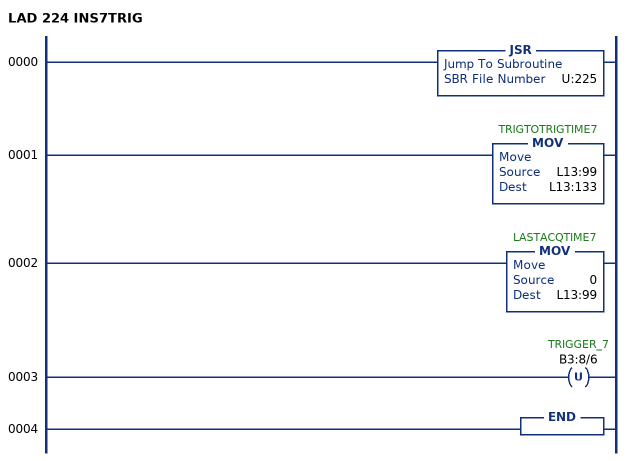
% Rung: 0 %
SOR JSR U:225 EOR
% Rung: 1 %
SOR MOV L13:99 L13:133 EOR
%   L13:99  LASTACQTIME7 %
%   L13:133  TRIGTOTRIGTIME7 %
% Rung: 2 %
SOR MOV 0 L13:99 EOR
%   L13:99  LASTACQTIME7 %
% Rung: 3 %
SOR OTU B3:8/6 EOR
%   B3:8/6  TRIGGER_7 %
% Rung: 4 %
SOR END EOR

LADDER 225 "FIFO7SET"
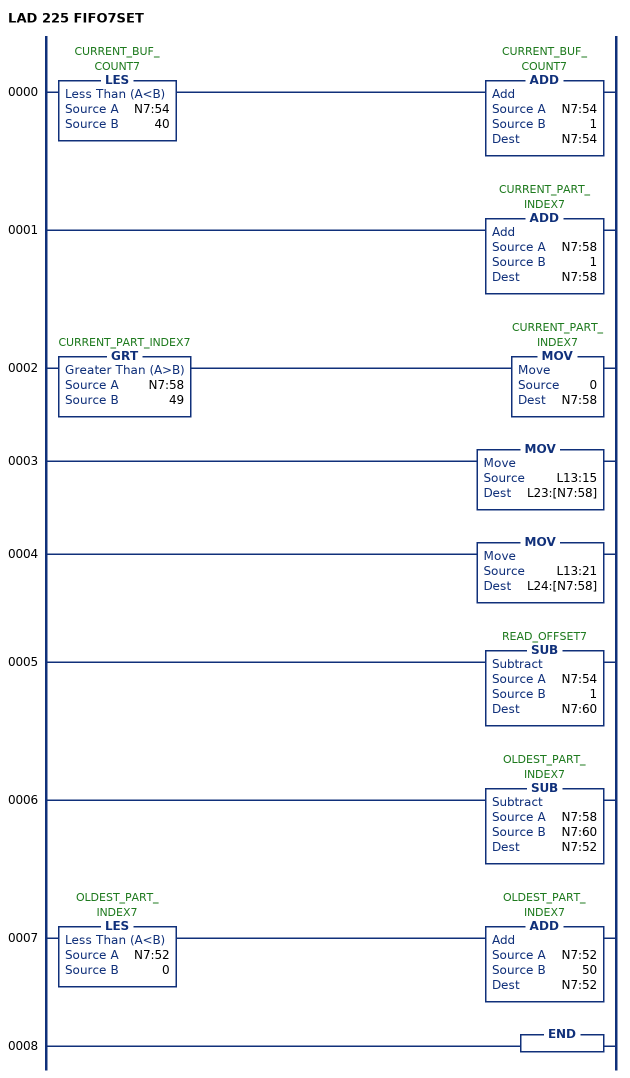
% Rung: 0 %
SOR LES N7:54 40 ADD N7:54 1 N7:54 EOR
%   N7:54  CURRENT_BUF_COUNT7 %
% Rung: 1 %
SOR ADD N7:58 1 N7:58 EOR
%   N7:58  CURRENT_PART_INDEX7 %
% Rung: 2 %
SOR GRT N7:58 49 MOV 0 N7:58 EOR
%   N7:58  CURRENT_PART_INDEX7 %
% Rung: 3 %
SOR MOV L13:15 L23:[N7:58] EOR
%   L13:15  TOP_TIME %
%   N7:58  CURRENT_PART_INDEX7 %
% Rung: 4 %
SOR MOV L13:21 L24:[N7:58] EOR
%   L13:21  TOP_POSITION %
%   N7:58  CURRENT_PART_INDEX7 %
% Rung: 5 %
SOR SUB N7:54 1 N7:60 EOR
%   N7:54  CURRENT_BUF_COUNT7 %
%   N7:60  READ_OFFSET7 %
% Rung: 6 %
SOR SUB N7:58 N7:60 N7:52 EOR
%   N7:58  CURRENT_PART_INDEX7 %
%   N7:60  READ_OFFSET7 %
%   N7:52  OLDEST_PART_INDEX7 %
% Rung: 7 %
SOR LES N7:52 0 ADD N7:52 50 N7:52 EOR
%   N7:52  OLDEST_PART_INDEX7 %
% Rung: 8 %
SOR END EOR

LADDER 226 "FIFO7GET"
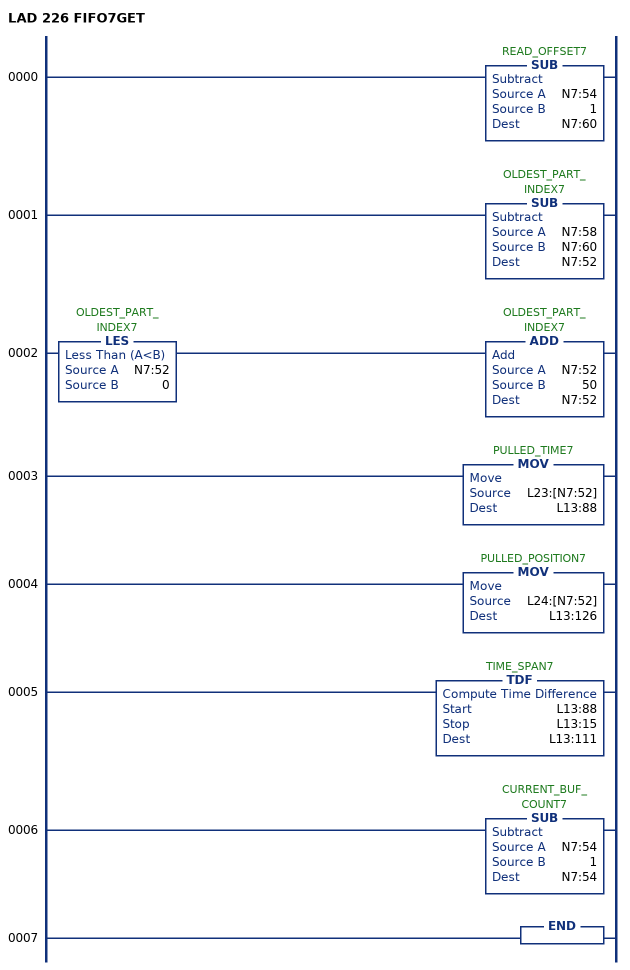
% Rung: 0 %
SOR SUB N7:54 1 N7:60 EOR
%   N7:54  CURRENT_BUF_COUNT7 %
%   N7:60  READ_OFFSET7 %
% Rung: 1 %
SOR SUB N7:58 N7:60 N7:52 EOR
%   N7:58  CURRENT_PART_INDEX7 %
%   N7:60  READ_OFFSET7 %
%   N7:52  OLDEST_PART_INDEX7 %
% Rung: 2 %
SOR LES N7:52 0 ADD N7:52 50 N7:52 EOR
%   N7:52  OLDEST_PART_INDEX7 %
% Rung: 3 %
SOR MOV L23:[N7:52] L13:88 EOR
%   N7:52  OLDEST_PART_INDEX7 %
%   L13:88  PULLED_TIME7 %
% Rung: 4 %
SOR MOV L24:[N7:52] L13:126 EOR
%   N7:52  OLDEST_PART_INDEX7 %
%   L13:126  PULLED_POSITION7 %
% Rung: 5 %
SOR TDF L13:88 L13:15 L13:111 EOR
%   L13:88  PULLED_TIME7 %
%   L13:15  TOP_TIME %
%   L13:111  TIME_SPAN7 %
% Rung: 6 %
SOR SUB N7:54 1 N7:54 EOR
%   N7:54  CURRENT_BUF_COUNT7 %
% Rung: 7 %
SOR END EOR

LADDER 227 "INSDATA7"
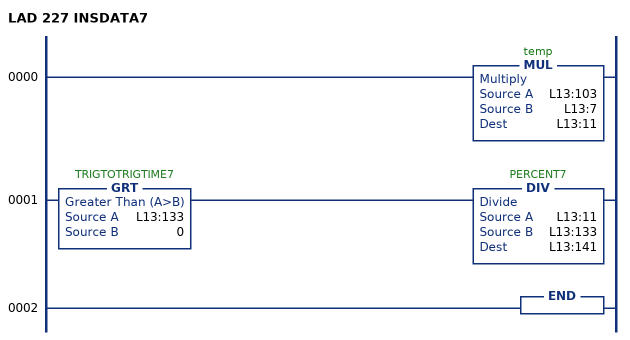
% Rung: 0 %
SOR MUL L13:103 L13:7 L13:11 EOR
%   L13:103  PROCESSTIME7 %
%   L13:7  PERCENT_MULTIPLYER %
%   L13:11  "temp" %
% Rung: 1 %
SOR GRT L13:133 0 DIV L13:11 L13:133 L13:141 EOR
%   L13:133  TRIGTOTRIGTIME7 %
%   L13:11  "temp" %
%   L13:141  PERCENT7 %
% Rung: 2 %
SOR END EOR

LADDER 228 "TESTFAULT7"
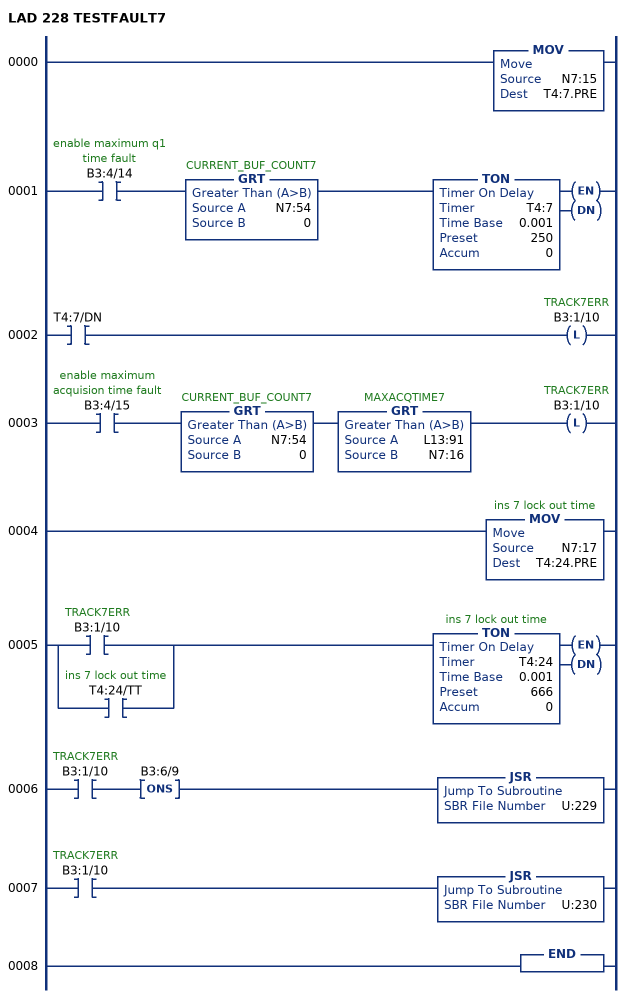
% Rung: 0 %
SOR MOV N7:15 T4:7.PRE EOR
%   N7:15  "max allowed ms time for q to be above 1 if safe fault is used" %
% Rung: 1 %
SOR XIC B3:4/14 GRT N7:54 0 TON T4:7 0.001 250 0 EOR
%   B3:4/14  "enable maximum q1 time fault" %
%   N7:54  CURRENT_BUF_COUNT7 %
% Rung: 2 %
SOR XIC T4:7/DN OTL B3:1/10 EOR
%   B3:1/10  TRACK7ERR %
% Rung: 3 %
SOR XIC B3:4/15 GRT N7:54 0 GRT L13:91 N7:16 OTL B3:1/10 EOR
%   B3:4/15  "enable maximum acquision time fault" %
%   N7:54  CURRENT_BUF_COUNT7 %
%   L13:91  MAXACQTIME7 %
%   N7:16  ACQUIRE_TIME_LIMIT  "maximum of the longest acquire time allowed if maximum acquire time fault is enabled" %
%   B3:1/10  TRACK7ERR %
% Rung: 4 %
SOR MOV N7:17 T4:24.PRE EOR
%   N7:17  "ms time setting to lock out inspection to give all pending images a chance to clear" %
%   T4:24  "ins 7 lock out time" %
% Rung: 5 %
SOR BST XIC B3:1/10 NXB XIC T4:24/TT BND TON T4:24 0.001 666 0 EOR
%   B3:1/10  TRACK7ERR %
%   T4:24  "ins 7 lock out time" %
% Rung: 6 %
SOR XIC B3:1/10 ONS B3:6/9 JSR U:229 EOR
%   B3:1/10  TRACK7ERR %
% Rung: 7 %
SOR XIC B3:1/10 JSR U:230 EOR
%   B3:1/10  TRACK7ERR %
% Rung: 8 %
SOR END EOR

LADDER 229 "INS7FIX1"
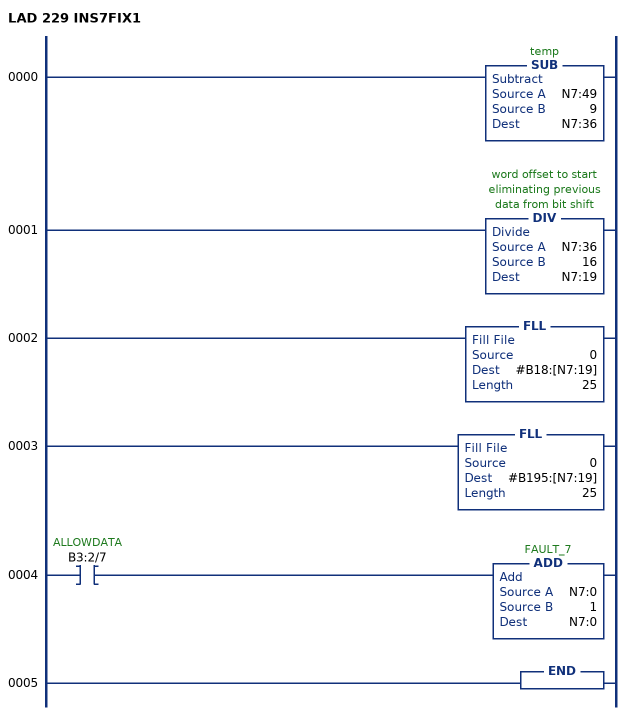
% Rung: 0 %
SOR SUB N7:49 9 N7:36 EOR
%   N7:49  INS_7_TRIG_LOC %
%   N7:36  "temp" %
% Rung: 1 %
SOR DIV N7:36 16 N7:19 EOR
%   N7:36  "temp" %
%   N7:19  "word offset to start eliminating previous data from bit shift" %
% Rung: 2 %
SOR FLL 0 #B18:[N7:19] 25 EOR
%   N7:19  "word offset to start eliminating previous data from bit shift" %
% Rung: 3 %
SOR FLL 0 #B195:[N7:19] 25 EOR
%   N7:19  "word offset to start eliminating previous data from bit shift" %
% Rung: 4 %
SOR XIC B3:2/7 ADD N7:0 1 N7:0 EOR
%   B3:2/7  ALLOWDATA %
%   N7:0  FAULT_7 %
% Rung: 5 %
SOR END EOR

LADDER 230 "INS7FIX2"
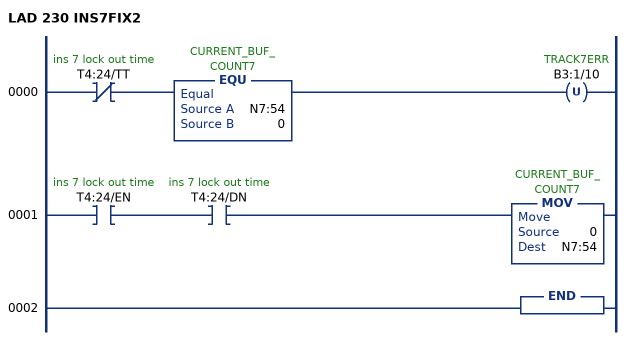
% Rung: 0 %
SOR XIO T4:24/TT EQU N7:54 0 OTU B3:1/10 EOR
%   T4:24  "ins 7 lock out time" %
%   N7:54  CURRENT_BUF_COUNT7 %
%   B3:1/10  TRACK7ERR %
% Rung: 1 %
SOR XIC T4:24/EN XIC T4:24/DN MOV 0 N7:54 EOR
%   T4:24  "ins 7 lock out time" %
%   N7:54  CURRENT_BUF_COUNT7 %
% Rung: 2 %
SOR END EOR

LADDER 232 "INS8"
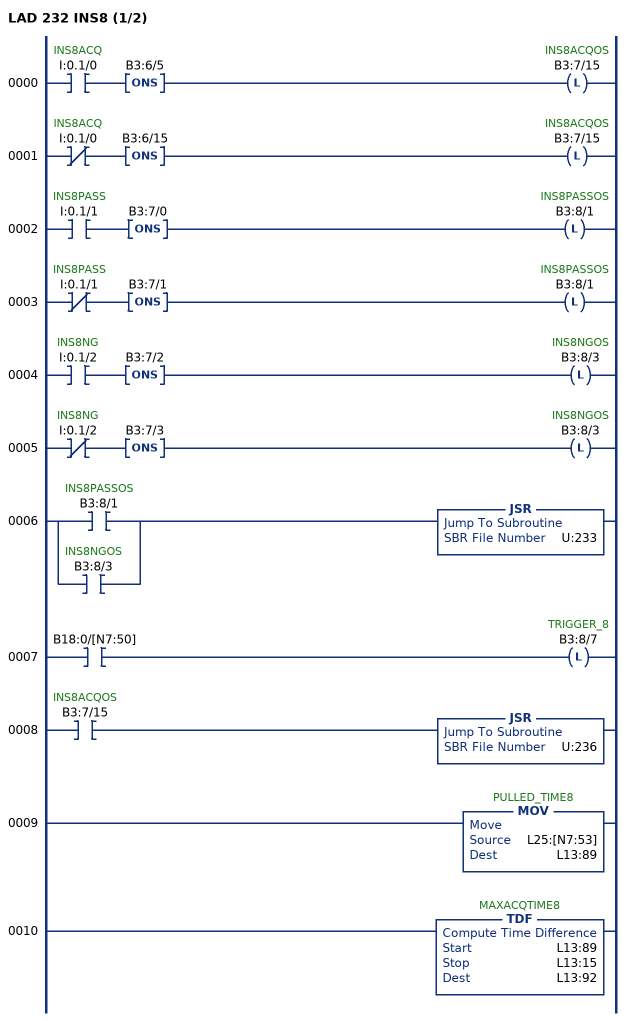
% Rung: 0 %
SOR XIC I:0.1/0 ONS B3:6/5 OTL B3:7/15 EOR
%   I:0.1/0  INS8ACQ %
%   B3:7/15  INS8ACQOS %
% Rung: 1 %
SOR XIO I:0.1/0 ONS B3:6/15 OTL B3:7/15 EOR
%   I:0.1/0  INS8ACQ %
%   B3:7/15  INS8ACQOS %
% Rung: 2 %
SOR XIC I:0.1/1 ONS B3:7/0 OTL B3:8/1 EOR
%   I:0.1/1  INS8PASS %
%   B3:8/1  INS8PASSOS %
% Rung: 3 %
SOR XIO I:0.1/1 ONS B3:7/1 OTL B3:8/1 EOR
%   I:0.1/1  INS8PASS %
%   B3:8/1  INS8PASSOS %
% Rung: 4 %
SOR XIC I:0.1/2 ONS B3:7/2 OTL B3:8/3 EOR
%   I:0.1/2  INS8NG %
%   B3:8/3  INS8NGOS %
% Rung: 5 %
SOR XIO I:0.1/2 ONS B3:7/3 OTL B3:8/3 EOR
%   I:0.1/2  INS8NG %
%   B3:8/3  INS8NGOS %
% Rung: 6 %
SOR BST XIC B3:8/1 NXB XIC B3:8/3 BND JSR U:233 EOR
%   B3:8/1  INS8PASSOS %
%   B3:8/3  INS8NGOS %
% Rung: 7 %
SOR XIC B18:0/[N7:50] OTL B3:8/7 EOR
%   B18:0  TOP_G %
%   N7:50  INS_8_TRIG_LOC %
%   B3:8/7  TRIGGER_8 %
% Rung: 8 %
SOR XIC B3:7/15 JSR U:236 EOR
%   B3:7/15  INS8ACQOS %
% Rung: 9 %
SOR MOV L25:[N7:53] L13:89 EOR
%   N7:53  OLDEST_PART_INDEX8 %
%   L13:89  PULLED_TIME8 %
% Rung: 10 %
SOR TDF L13:89 L13:15 L13:92 EOR
%   L13:89  PULLED_TIME8 %
%   L13:15  TOP_TIME %
%   L13:92  MAXACQTIME8 %

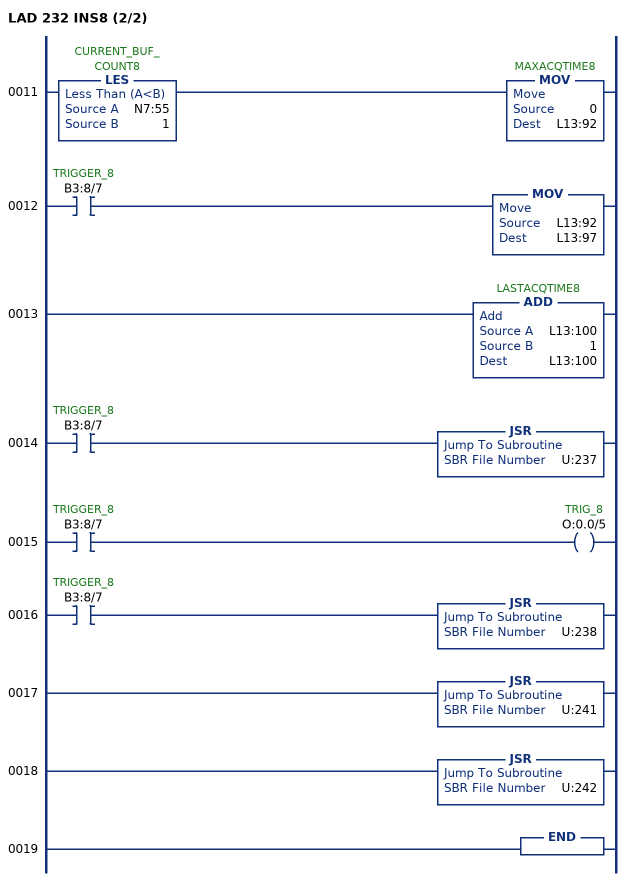
% Rung: 11 %
SOR LES N7:55 1 MOV 0 L13:92 EOR
%   N7:55  CURRENT_BUF_COUNT8 %
%   L13:92  MAXACQTIME8 %
% Rung: 12 %
SOR XIC B3:8/7 MOV L13:92 L13:97 EOR
%   B3:8/7  TRIGGER_8 %
%   L13:92  MAXACQTIME8 %
% Rung: 13 %
SOR ADD L13:100 1 L13:100 EOR
%   L13:100  LASTACQTIME8 %
% Rung: 14 %
SOR XIC B3:8/7 JSR U:237 EOR
%   B3:8/7  TRIGGER_8 %
% Rung: 15 %
SOR XIC B3:8/7 OTE O:0.0/5 EOR
%   B3:8/7  TRIGGER_8 %
%   O:0.0/5  TRIG_8 %
% Rung: 16 %
SOR XIC B3:8/7 JSR U:238 EOR
%   B3:8/7  TRIGGER_8 %
% Rung: 17 %
SOR JSR U:241 EOR
% Rung: 18 %
SOR JSR U:242 EOR
% Rung: 19 %
SOR END EOR

LADDER 233 "INS8RESULT"
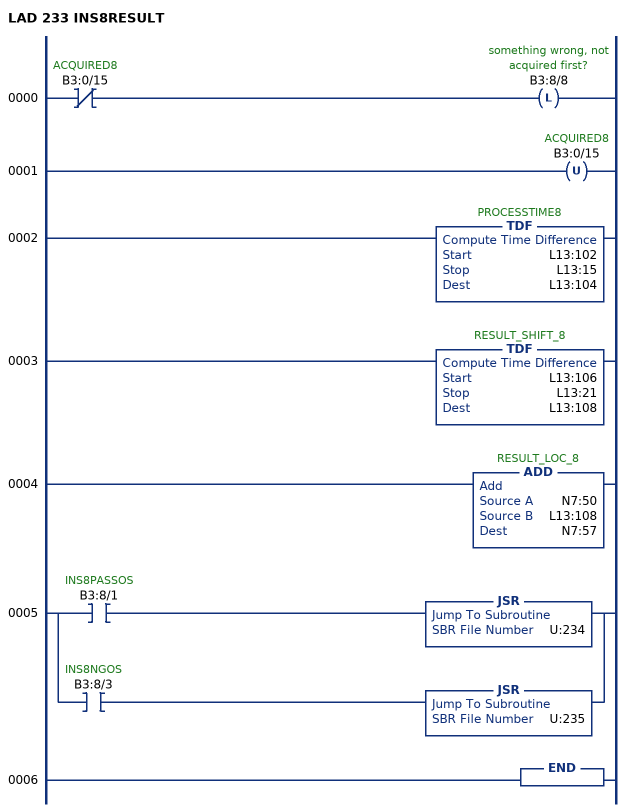
% Rung: 0 %
SOR XIO B3:0/15 OTL B3:8/8 EOR
%   B3:0/15  ACQUIRED8 %
%   B3:8/8  "something wrong, not acquired first?" %
% Rung: 1 %
SOR OTU B3:0/15 EOR
%   B3:0/15  ACQUIRED8 %
% Rung: 2 %
SOR TDF L13:102 L13:15 L13:104 EOR
%   L13:102  TIMEOFACQ8 %
%   L13:15  TOP_TIME %
%   L13:104  PROCESSTIME8 %
% Rung: 3 %
SOR TDF L13:106 L13:21 L13:108 EOR
%   L13:106  PROCESS_START_POS_8 %
%   L13:21  TOP_POSITION %
%   L13:108  RESULT_SHIFT_8 %
% Rung: 4 %
SOR ADD N7:50 L13:108 N7:57 EOR
%   N7:50  INS_8_TRIG_LOC %
%   L13:108  RESULT_SHIFT_8 %
%   N7:57  RESULT_LOC_8 %
% Rung: 5 %
SOR BST XIC B3:8/1 JSR U:234 NXB XIC B3:8/3 JSR U:235 BND EOR
%   B3:8/1  INS8PASSOS %
%   B3:8/3  INS8NGOS %
% Rung: 6 %
SOR END EOR

LADDER 234 "INS8PASS"
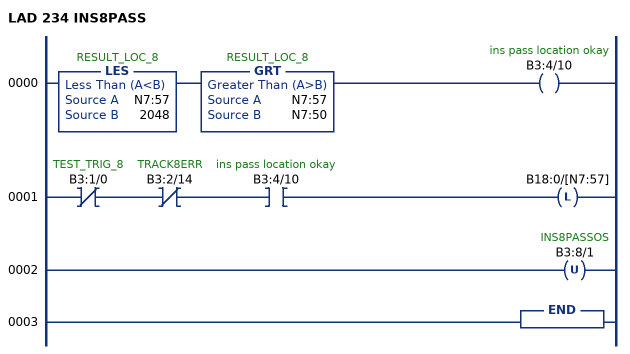
% Rung: 0 %
SOR LES N7:57 2048 GRT N7:57 N7:50 OTE B3:4/10 EOR
%   N7:57  RESULT_LOC_8 %
%   N7:50  INS_8_TRIG_LOC %
%   B3:4/10  "ins pass location okay" %
% Rung: 1 %
SOR XIO B3:1/0 XIO B3:2/14 XIC B3:4/10 OTL B18:0/[N7:57] EOR
%   B3:1/0  TEST_TRIG_8 %
%   B3:2/14  TRACK8ERR %
%   B3:4/10  "ins pass location okay" %
%   B18:0  TOP_G %
%   N7:57  RESULT_LOC_8 %
% Rung: 2 %
SOR OTU B3:8/1 EOR
%   B3:8/1  INS8PASSOS %
% Rung: 3 %
SOR END EOR

LADDER 235 "INS8FAIL"
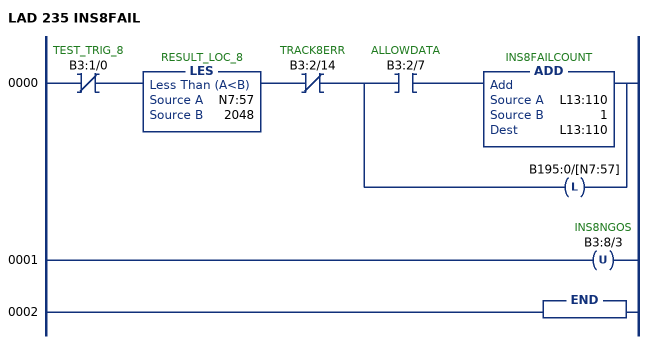
% Rung: 0 %
SOR XIO B3:1/0 LES N7:57 2048 XIO B3:2/14 BST XIC B3:2/7 ADD L13:110 1 L13:110 NXB OTL B195:0/[N7:57] BND EOR
%   B3:1/0  TEST_TRIG_8 %
%   N7:57  RESULT_LOC_8 %
%   B3:2/14  TRACK8ERR %
%   B3:2/7  ALLOWDATA %
%   L13:110  INS8FAILCOUNT %
%   B195:0  TOP_NG %
% Rung: 1 %
SOR OTU B3:8/3 EOR
%   B3:8/3  INS8NGOS %
% Rung: 2 %
SOR END EOR

LADDER 236 "INS8ACQ"
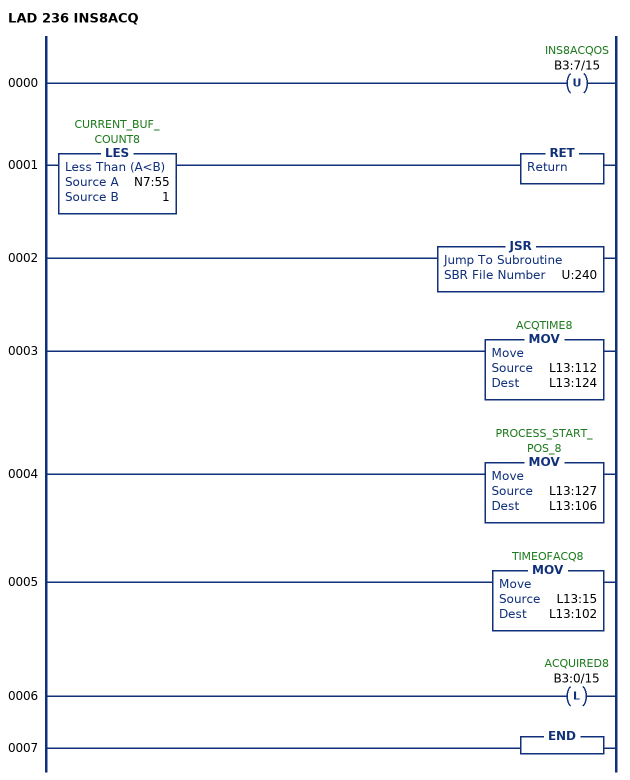
% Rung: 0 %
SOR OTU B3:7/15 EOR
%   B3:7/15  INS8ACQOS %
% Rung: 1 %
SOR LES N7:55 1 RET EOR
%   N7:55  CURRENT_BUF_COUNT8 %
% Rung: 2 %
SOR JSR U:240 EOR
% Rung: 3 %
SOR MOV L13:112 L13:124 EOR
%   L13:112  TIME_SPAN8 %
%   L13:124  ACQTIME8 %
% Rung: 4 %
SOR MOV L13:127 L13:106 EOR
%   L13:127  PULLED_POSITION8 %
%   L13:106  PROCESS_START_POS_8 %
% Rung: 5 %
SOR MOV L13:15 L13:102 EOR
%   L13:15  TOP_TIME %
%   L13:102  TIMEOFACQ8 %
% Rung: 6 %
SOR OTL B3:0/15 EOR
%   B3:0/15  ACQUIRED8 %
% Rung: 7 %
SOR END EOR

LADDER 237 "Q8TIMETEST"
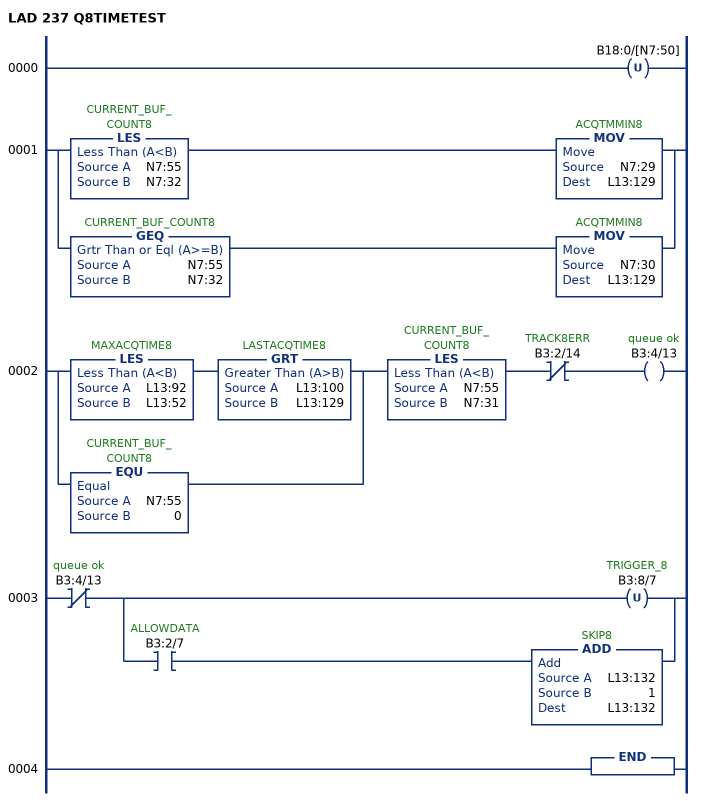
% Rung: 0 %
SOR OTU B18:0/[N7:50] EOR
%   B18:0  TOP_G %
%   N7:50  INS_8_TRIG_LOC %
% Rung: 1 %
SOR BST LES N7:55 N7:32 MOV N7:29 L13:129 NXB GEQ N7:55 N7:32 MOV N7:30 L13:129 BND EOR
%   N7:55  CURRENT_BUF_COUNT8 %
%   N7:32  BUF_CAM_LIMIT %
%   N7:29  CAM_BUF_ACQ_TM %
%   L13:129  ACQTMMIN8 %
%   N7:30  PC_BUF_ACQ_TM %
% Rung: 2 %
SOR BST LES L13:92 L13:52 GRT L13:100 L13:129 NXB EQU N7:55 0 BND LES N7:55 N7:31 XIO B3:2/14 OTE B3:4/13 EOR
%   L13:92  MAXACQTIME8 %
%   L13:52  ACQTIMELIMIT %
%   L13:100  LASTACQTIME8 %
%   L13:129  ACQTMMIN8 %
%   N7:55  CURRENT_BUF_COUNT8 %
%   N7:31  MAX_BUFF_CT  "maximum buffers" %
%   B3:2/14  TRACK8ERR %
%   B3:4/13  "queue ok" %
% Rung: 3 %
SOR XIO B3:4/13 BST OTU B3:8/7 NXB XIC B3:2/7 ADD L13:132 1 L13:132 BND EOR
%   B3:4/13  "queue ok" %
%   B3:8/7  TRIGGER_8 %
%   B3:2/7  ALLOWDATA %
%   L13:132  SKIP8 %
% Rung: 4 %
SOR END EOR

LADDER 238 "INS8TRIG"
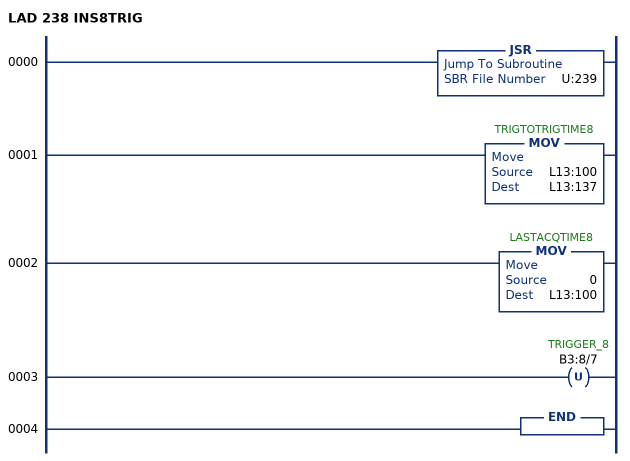
% Rung: 0 %
SOR JSR U:239 EOR
% Rung: 1 %
SOR MOV L13:100 L13:137 EOR
%   L13:100  LASTACQTIME8 %
%   L13:137  TRIGTOTRIGTIME8 %
% Rung: 2 %
SOR MOV 0 L13:100 EOR
%   L13:100  LASTACQTIME8 %
% Rung: 3 %
SOR OTU B3:8/7 EOR
%   B3:8/7  TRIGGER_8 %
% Rung: 4 %
SOR END EOR

LADDER 239 "FIFO8SET"
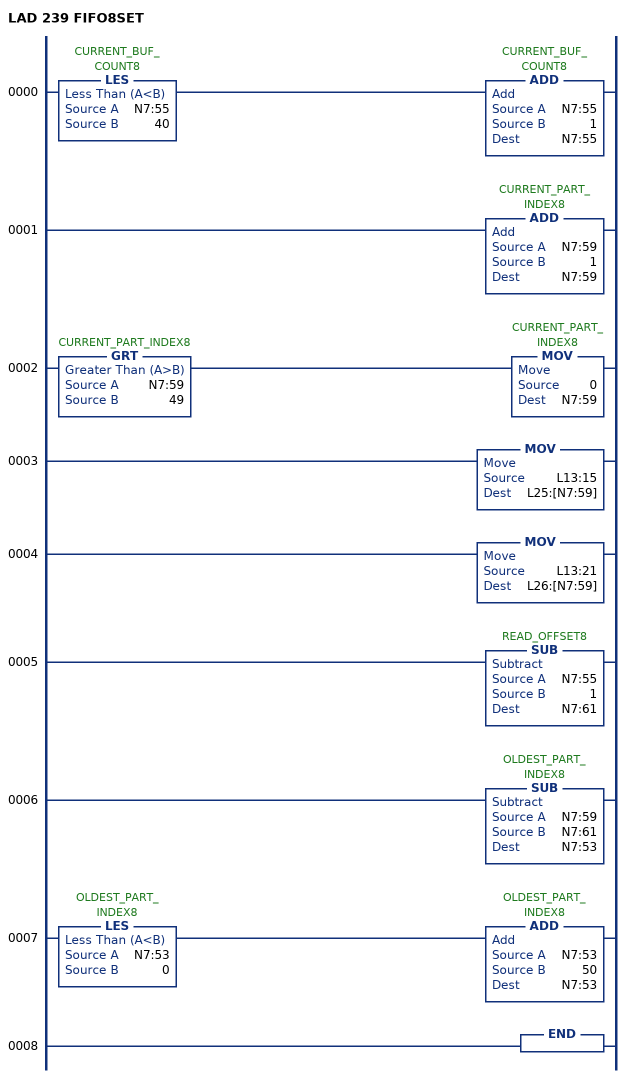
% Rung: 0 %
SOR LES N7:55 40 ADD N7:55 1 N7:55 EOR
%   N7:55  CURRENT_BUF_COUNT8 %
% Rung: 1 %
SOR ADD N7:59 1 N7:59 EOR
%   N7:59  CURRENT_PART_INDEX8 %
% Rung: 2 %
SOR GRT N7:59 49 MOV 0 N7:59 EOR
%   N7:59  CURRENT_PART_INDEX8 %
% Rung: 3 %
SOR MOV L13:15 L25:[N7:59] EOR
%   L13:15  TOP_TIME %
%   N7:59  CURRENT_PART_INDEX8 %
% Rung: 4 %
SOR MOV L13:21 L26:[N7:59] EOR
%   L13:21  TOP_POSITION %
%   N7:59  CURRENT_PART_INDEX8 %
% Rung: 5 %
SOR SUB N7:55 1 N7:61 EOR
%   N7:55  CURRENT_BUF_COUNT8 %
%   N7:61  READ_OFFSET8 %
% Rung: 6 %
SOR SUB N7:59 N7:61 N7:53 EOR
%   N7:59  CURRENT_PART_INDEX8 %
%   N7:61  READ_OFFSET8 %
%   N7:53  OLDEST_PART_INDEX8 %
% Rung: 7 %
SOR LES N7:53 0 ADD N7:53 50 N7:53 EOR
%   N7:53  OLDEST_PART_INDEX8 %
% Rung: 8 %
SOR END EOR

LADDER 240 "FIFO8GET"
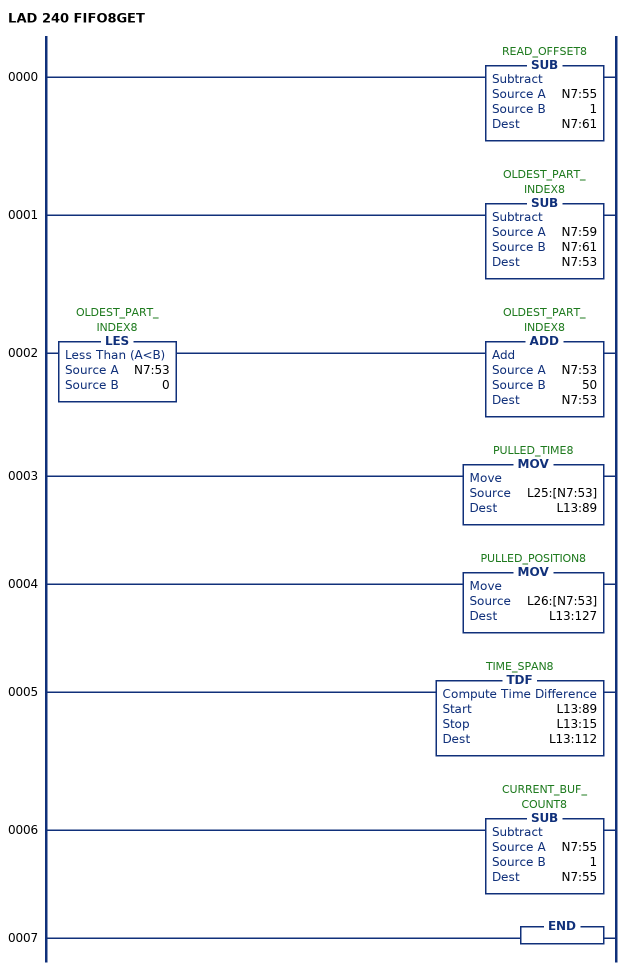
% Rung: 0 %
SOR SUB N7:55 1 N7:61 EOR
%   N7:55  CURRENT_BUF_COUNT8 %
%   N7:61  READ_OFFSET8 %
% Rung: 1 %
SOR SUB N7:59 N7:61 N7:53 EOR
%   N7:59  CURRENT_PART_INDEX8 %
%   N7:61  READ_OFFSET8 %
%   N7:53  OLDEST_PART_INDEX8 %
% Rung: 2 %
SOR LES N7:53 0 ADD N7:53 50 N7:53 EOR
%   N7:53  OLDEST_PART_INDEX8 %
% Rung: 3 %
SOR MOV L25:[N7:53] L13:89 EOR
%   N7:53  OLDEST_PART_INDEX8 %
%   L13:89  PULLED_TIME8 %
% Rung: 4 %
SOR MOV L26:[N7:53] L13:127 EOR
%   N7:53  OLDEST_PART_INDEX8 %
%   L13:127  PULLED_POSITION8 %
% Rung: 5 %
SOR TDF L13:89 L13:15 L13:112 EOR
%   L13:89  PULLED_TIME8 %
%   L13:15  TOP_TIME %
%   L13:112  TIME_SPAN8 %
% Rung: 6 %
SOR SUB N7:55 1 N7:55 EOR
%   N7:55  CURRENT_BUF_COUNT8 %
% Rung: 7 %
SOR END EOR

LADDER 241 "INSDATA8"
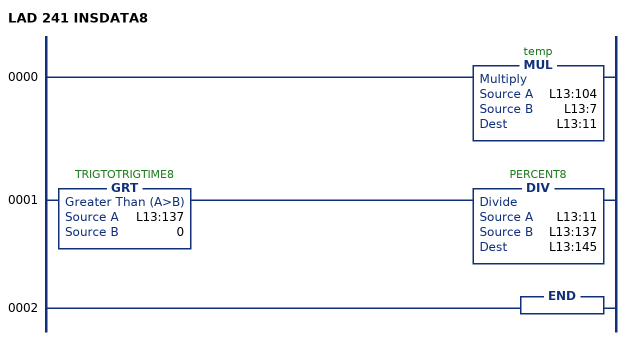
% Rung: 0 %
SOR MUL L13:104 L13:7 L13:11 EOR
%   L13:104  PROCESSTIME8 %
%   L13:7  PERCENT_MULTIPLYER %
%   L13:11  "temp" %
% Rung: 1 %
SOR GRT L13:137 0 DIV L13:11 L13:137 L13:145 EOR
%   L13:137  TRIGTOTRIGTIME8 %
%   L13:11  "temp" %
%   L13:145  PERCENT8 %
% Rung: 2 %
SOR END EOR

LADDER 242 "TESTFAULT8"
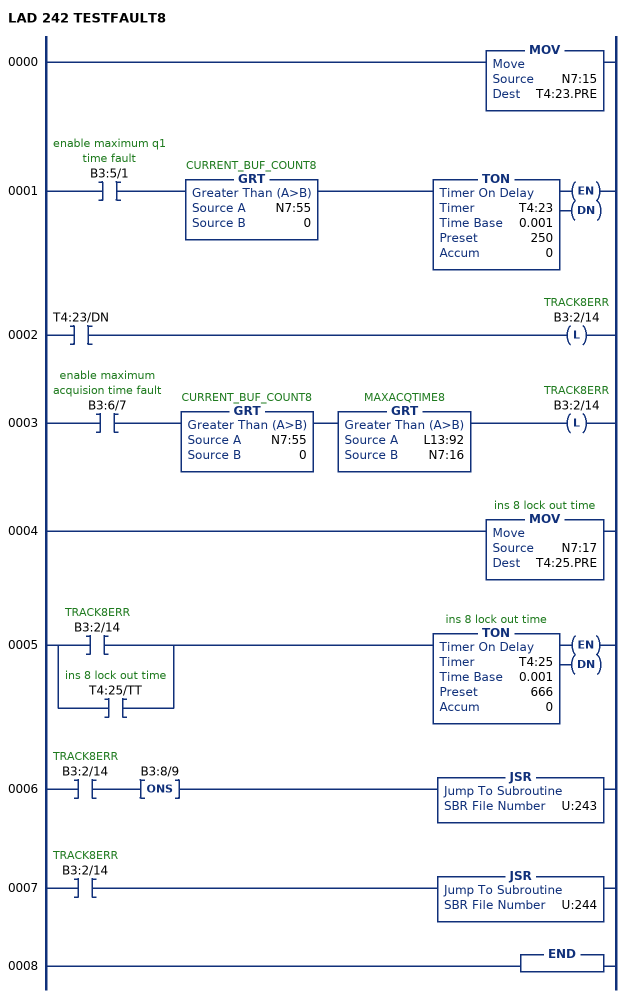
% Rung: 0 %
SOR MOV N7:15 T4:23.PRE EOR
%   N7:15  "max allowed ms time for q to be above 1 if safe fault is used" %
% Rung: 1 %
SOR XIC B3:5/1 GRT N7:55 0 TON T4:23 0.001 250 0 EOR
%   B3:5/1  "enable maximum q1 time fault" %
%   N7:55  CURRENT_BUF_COUNT8 %
% Rung: 2 %
SOR XIC T4:23/DN OTL B3:2/14 EOR
%   B3:2/14  TRACK8ERR %
% Rung: 3 %
SOR XIC B3:6/7 GRT N7:55 0 GRT L13:92 N7:16 OTL B3:2/14 EOR
%   B3:6/7  "enable maximum acquision time fault" %
%   N7:55  CURRENT_BUF_COUNT8 %
%   L13:92  MAXACQTIME8 %
%   N7:16  ACQUIRE_TIME_LIMIT  "maximum of the longest acquire time allowed if maximum acquire time fault is enabled" %
%   B3:2/14  TRACK8ERR %
% Rung: 4 %
SOR MOV N7:17 T4:25.PRE EOR
%   N7:17  "ms time setting to lock out inspection to give all pending images a chance to clear" %
%   T4:25  "ins 8 lock out time" %
% Rung: 5 %
SOR BST XIC B3:2/14 NXB XIC T4:25/TT BND TON T4:25 0.001 666 0 EOR
%   B3:2/14  TRACK8ERR %
%   T4:25  "ins 8 lock out time" %
% Rung: 6 %
SOR XIC B3:2/14 ONS B3:8/9 JSR U:243 EOR
%   B3:2/14  TRACK8ERR %
% Rung: 7 %
SOR XIC B3:2/14 JSR U:244 EOR
%   B3:2/14  TRACK8ERR %
% Rung: 8 %
SOR END EOR

LADDER 243 "INS8FIX1"
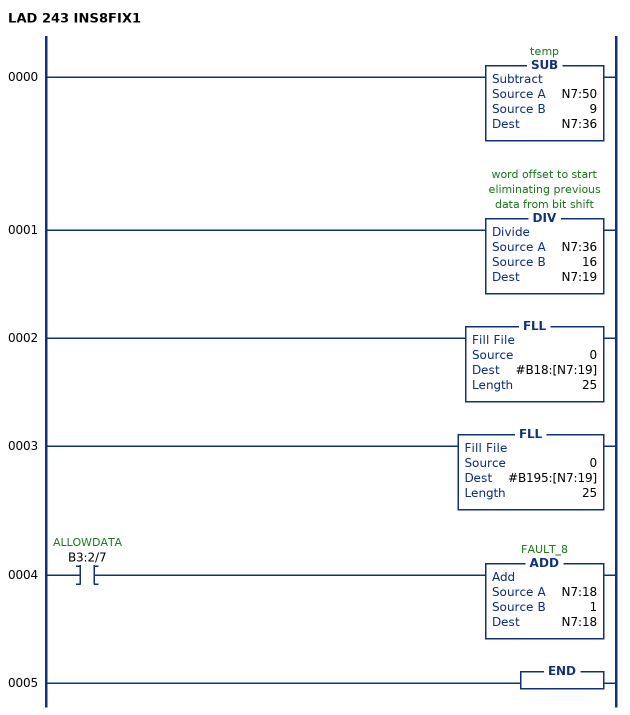
% Rung: 0 %
SOR SUB N7:50 9 N7:36 EOR
%   N7:50  INS_8_TRIG_LOC %
%   N7:36  "temp" %
% Rung: 1 %
SOR DIV N7:36 16 N7:19 EOR
%   N7:36  "temp" %
%   N7:19  "word offset to start eliminating previous data from bit shift" %
% Rung: 2 %
SOR FLL 0 #B18:[N7:19] 25 EOR
%   N7:19  "word offset to start eliminating previous data from bit shift" %
% Rung: 3 %
SOR FLL 0 #B195:[N7:19] 25 EOR
%   N7:19  "word offset to start eliminating previous data from bit shift" %
% Rung: 4 %
SOR XIC B3:2/7 ADD N7:18 1 N7:18 EOR
%   B3:2/7  ALLOWDATA %
%   N7:18  FAULT_8 %
% Rung: 5 %
SOR END EOR

LADDER 244 "INS8FIX2"
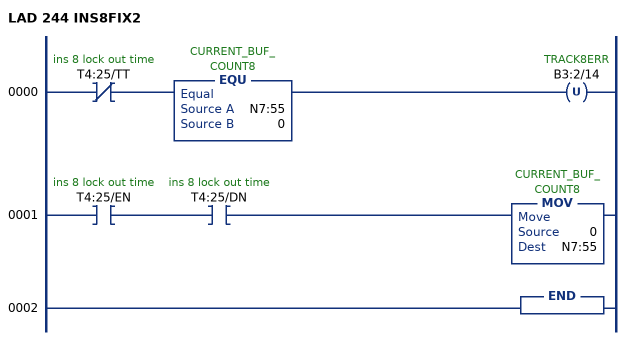
% Rung: 0 %
SOR XIO T4:25/TT EQU N7:55 0 OTU B3:2/14 EOR
%   T4:25  "ins 8 lock out time" %
%   N7:55  CURRENT_BUF_COUNT8 %
%   B3:2/14  TRACK8ERR %
% Rung: 1 %
SOR XIC T4:25/EN XIC T4:25/DN MOV 0 N7:55 EOR
%   T4:25  "ins 8 lock out time" %
%   N7:55  CURRENT_BUF_COUNT8 %
% Rung: 2 %
SOR END EOR

LADDER 249 "PASS BLOW"
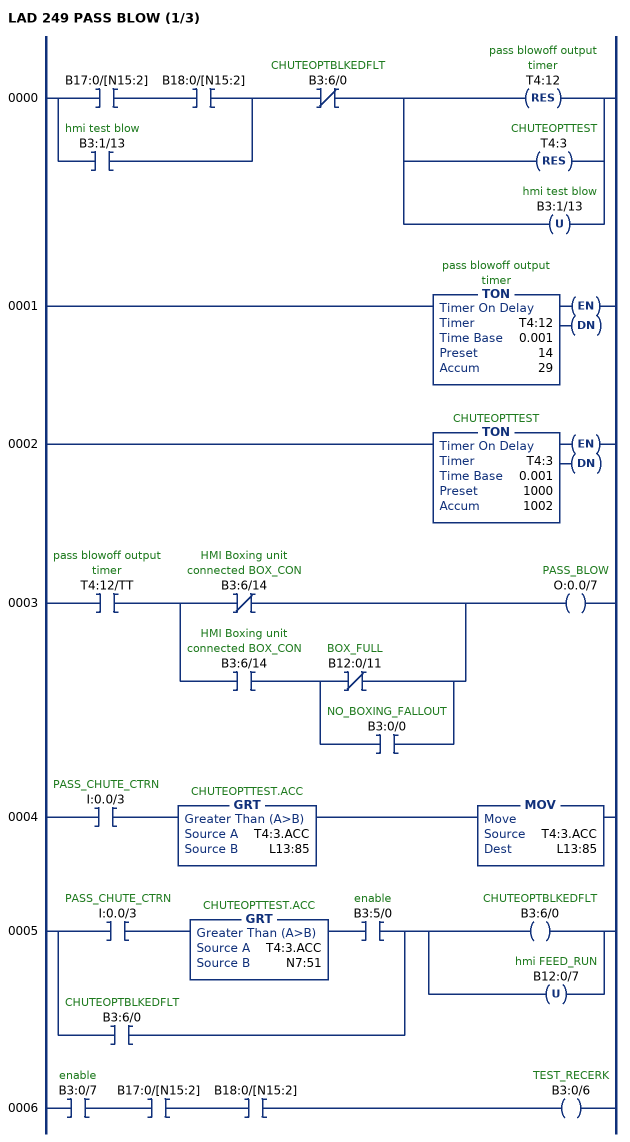
% Rung: 0 %
SOR BST XIC B17:0/[N15:2] XIC B18:0/[N15:2] NXB XIC B3:1/13 BND XIO B3:6/0 BST RES T4:12 NXB RES T4:3 NXB OTU B3:1/13 BND EOR
%   B17:0  SIDE_G %
%   N15:2  BLOW_PT %
%   B18:0  TOP_G %
%   B3:1/13  "hmi test blow" %
%   B3:6/0  CHUTEOPTBLKEDFLT %
%   T4:12  "pass blowoff output timer" %
%   T4:3  CHUTEOPTTEST %
% Rung: 1 %
SOR TON T4:12 0.001 14 29 EOR
%   T4:12  "pass blowoff output timer" %
% Rung: 2 %
SOR TON T4:3 0.001 1000 1002 EOR
%   T4:3  CHUTEOPTTEST %
% Rung: 3 %
SOR XIC T4:12/TT BST XIO B3:6/14 NXB XIC B3:6/14 BST XIO B12:0/11 NXB XIC B3:0/0 BND BND OTE O:0.0/7 EOR
%   T4:12  "pass blowoff output timer" %
%   B3:6/14  BOX_CON  "HMI Boxing unit connected" %
%   B12:0/11  BOX_FULL %
%   B3:0/0  NO_BOXING_FALLOUT %
%   O:0.0/7  PASS_BLOW %
% Rung: 4 %
SOR XIC I:0.0/3 GRT T4:3.ACC L13:85 MOV T4:3.ACC L13:85 EOR
%   I:0.0/3  PASS_CHUTE_CTRN %
%   T4:3  CHUTEOPTTEST %
% Rung: 5 %
SOR BST XIC I:0.0/3 GRT T4:3.ACC N7:51 XIC B3:5/0 NXB XIC B3:6/0 BND BST OTE B3:6/0 NXB OTU B12:0/7 BND EOR
%   I:0.0/3  PASS_CHUTE_CTRN %
%   T4:3  CHUTEOPTTEST %
%   B3:5/0  "enable" %
%   B3:6/0  CHUTEOPTBLKEDFLT %
%   B12:0/7  FEED_RUN  "hmi" %
% Rung: 6 %
SOR XIC B3:0/7 XIC B17:0/[N15:2] XIC B18:0/[N15:2] OTE B3:0/6 EOR
%   B3:0/7  "enable" %
%   B17:0  SIDE_G %
%   N15:2  BLOW_PT %
%   B18:0  TOP_G %
%   B3:0/6  TEST_RECERK %

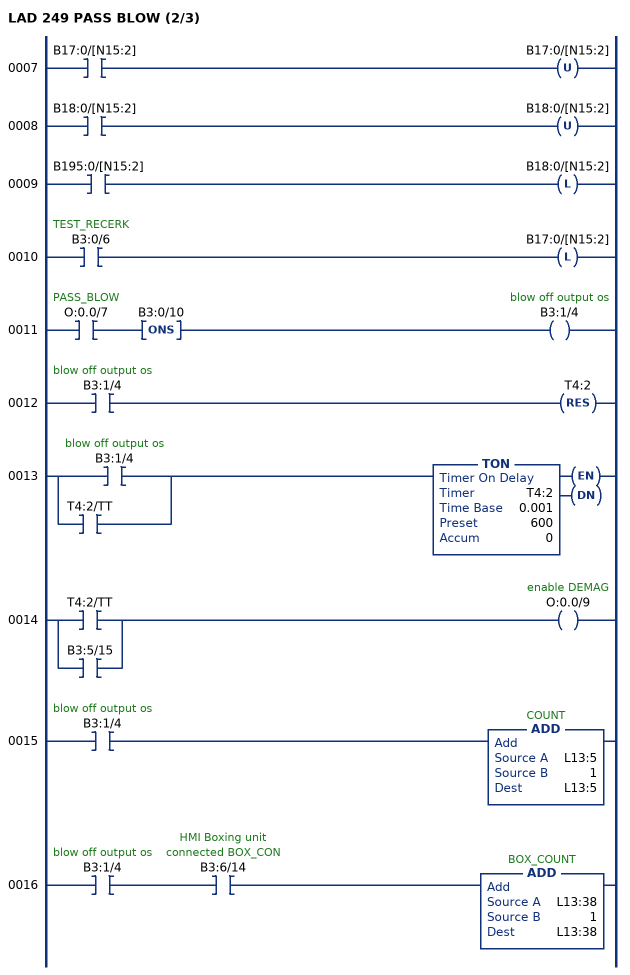
% Rung: 7 %
SOR XIC B17:0/[N15:2] OTU B17:0/[N15:2] EOR
%   B17:0  SIDE_G %
%   N15:2  BLOW_PT %
% Rung: 8 %
SOR XIC B18:0/[N15:2] OTU B18:0/[N15:2] EOR
%   B18:0  TOP_G %
%   N15:2  BLOW_PT %
% Rung: 9 %
SOR XIC B195:0/[N15:2] OTL B18:0/[N15:2] EOR
%   B195:0  TOP_NG %
%   N15:2  BLOW_PT %
%   B18:0  TOP_G %
% Rung: 10 %
SOR XIC B3:0/6 OTL B17:0/[N15:2] EOR
%   B3:0/6  TEST_RECERK %
%   B17:0  SIDE_G %
%   N15:2  BLOW_PT %
% Rung: 11 %
SOR XIC O:0.0/7 ONS B3:0/10 OTE B3:1/4 EOR
%   O:0.0/7  PASS_BLOW %
%   B3:1/4  "blow off output os" %
% Rung: 12 %
SOR XIC B3:1/4 RES T4:2 EOR
%   B3:1/4  "blow off output os" %
% Rung: 13 %
SOR BST XIC B3:1/4 NXB XIC T4:2/TT BND TON T4:2 0.001 600 0 EOR
%   B3:1/4  "blow off output os" %
% Rung: 14 %
SOR BST XIC T4:2/TT NXB XIC B3:5/15 BND OTE O:0.0/9 EOR
%   O:0.0/9  DEMAG  "enable" %
% Rung: 15 %
SOR XIC B3:1/4 ADD L13:5 1 L13:5 EOR
%   B3:1/4  "blow off output os" %
%   L13:5  COUNT %
% Rung: 16 %
SOR XIC B3:1/4 XIC B3:6/14 ADD L13:38 1 L13:38 EOR
%   B3:1/4  "blow off output os" %
%   B3:6/14  BOX_CON  "HMI Boxing unit connected" %
%   L13:38  BOX_COUNT %

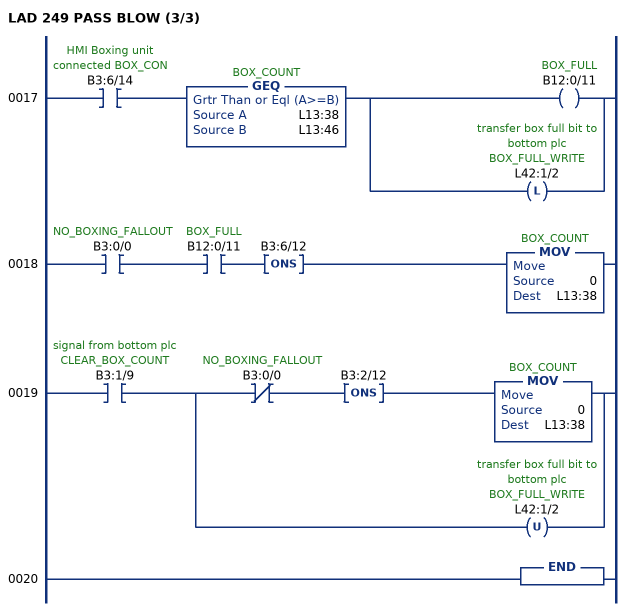
% Rung: 17 %
SOR XIC B3:6/14 GEQ L13:38 L13:46 BST OTE B12:0/11 NXB OTL L42:1/2 BND EOR
%   B3:6/14  BOX_CON  "HMI Boxing unit connected" %
%   L13:38  BOX_COUNT %
%   L13:46  BOX_LIMIT  "box count setpoint" %
%   B12:0/11  BOX_FULL %
%   L42:1/2  BOX_FULL_WRITE  "transfer box full bit to bottom plc" %
% Rung: 18 %
SOR XIC B3:0/0 XIC B12:0/11 ONS B3:6/12 MOV 0 L13:38 EOR
%   B3:0/0  NO_BOXING_FALLOUT %
%   B12:0/11  BOX_FULL %
%   L13:38  BOX_COUNT %
% Rung: 19 %
SOR XIC B3:1/9 BST XIO B3:0/0 ONS B3:2/12 MOV 0 L13:38 NXB OTU L42:1/2 BND EOR
%   B3:1/9  CLEAR_BOX_COUNT  "signal from bottom plc" %
%   B3:0/0  NO_BOXING_FALLOUT %
%   L13:38  BOX_COUNT %
%   L42:1/2  BOX_FULL_WRITE  "transfer box full bit to bottom plc" %
% Rung: 20 %
SOR END EOR

LADDER 250 "RECERK"
